FUNCTION_BLOCK BoolSub EXTENDS Object IMPLEMENTS I_BoolSub
VAR_OUTPUT
	Q: BOOL;
END_VAR
VAR
	_pub: I_BoolPub;
END_VAR

//Work in progress

METHOD Attach_Pub
VAR_INPUT
	IObject: I_SYS_COMP_Object;
END_VAR
VAR
	_pub: I_BoolPub;
END_VAR
END_METHOD

METHOD Remove_Pub
VAR_INPUT
	IObject: I_SYS_COMP_Object;
END_VAR
VAR
	_pub: I_BoolPub;
END_VAR
END_METHOD

PROPERTY Set : I_SYS_COMP_Object
SET
Q := Set;
END_SET
END_PROPERTY

END_FUNCTION_BLOCK

(* stored: Version 1.1.0.1, ProductVersion 3.1.4024.12
   POU BoolSub: Id {9a0adf1b-c06f-431b-bf2e-59f510babc3c}, SpecialFunc None
   Method Attach_Pub: Id {2b2b3796-f7a6-4f30-bc29-b9185adf24d2}
   Method Remove_Pub: Id {0e1de50b-acb7-4f7a-9249-575bc9972f3e}
   Property Set: Id {026c3244-79fa-4084-910f-e764ee859730}
   Set Set: Id {27b434e4-14dc-4193-a92a-29fa9744b8db} *)
